(* IEC 61131-3 sources: AXOpen/src/components.festo.drives/ctrl/src/AxoCmmtAs (part 3) *)

                        MC_TorqueControlPositionLimit_PV :=  PositionLimit;
                        MC_TorqueControlVelocity_PV      :=  Velocity;
                        MC_TorqueControlAcceleration_PV  :=  Acceleration;
                        MC_TorqueControlDeceleration_PV  :=  Deceleration;
                        MC_TorqueControlJerk_PV          :=  Jerk;
                        MC_TorqueControlDirection_PV     :=  Direction;
                        MC_TorqueControlTorque_PV        :=  Torque;
                        MC_TorqueControlTorqueRamp_PV    :=  TorqueRamp;
                        State := UINT#120;
                    END_IF;
                END_IF;
                IF State = UINT#120 THEN
                    Busy := TRUE;
                    Active := TRUE;
                    IF MC_TorqueControlPositiveDirectionA AND THIS.ActualPosition >= MC_TorqueControlPositionLimit_PV THEN
                        State := UINT#129;
                        Messenger.Activate(         UINT#1538, eAxoMessageCategory#ProgrammingError);
                        MC_TorqueControlErrorID :=  DINT#1538;
                    ELSIF NOT MC_TorqueControlPositiveDirectionA AND THIS.ActualPosition <= MC_TorqueControlPositionLimit_PV THEN
                        State := UINT#129;
                        Messenger.Activate(         UINT#1539, eAxoMessageCategory#ProgrammingError);
                        MC_TorqueControlErrorID :=  DINT#1539;
                    ELSE
                        State := UINT#121;
                    END_IF;
                END_IF;
                //Writing PNU 12168 Clamping torque
                IF State = UINT#121 THEN
                    Busy := TRUE;
                    Active := TRUE;
                    Parametrization.Inputs.Enable := TRUE;
                    Parametrization.Inputs.ReadWrite   := TRUE;
                    Parametrization.Inputs.ParameterNo := 12168;
                    Parametrization.Inputs.Subindex    := 0;
                    Parametrization.Inputs.AxisNo  := BYTE#1;
                    Parametrization.Inputs.HardwareId  := _AxisReference^.HWIDs.HW_ModuleAccessPoint;
                    Parametrization.Inputs.ValueWriteREAL := TO_REAL(MC_TorqueControlTorque_PV * ScalingConstantRequiredTorque);
                    IF Parametrization.Outputs.Done AND NOT Parametrization.Outputs.Error THEN
                        Parametrization.Inputs.Enable := FALSE;
                        Parametrization.Inputs.ReadWrite   := FALSE;
                        State := UINT#122;
                        RETURN;
                    END_IF;
                    IF Parametrization.Outputs.Error THEN
                        Messenger.Activate(         UINT#1540, eAxoMessageCategory#Error);
                        MC_TorqueControlErrorID :=  DINT#1540;
                        Parametrization.Inputs.Enable := FALSE;
                        Parametrization.Inputs.ReadWrite   := FALSE;
                        State := UINT#129;
                    END_IF;
                END_IF;
                //Writing PNU 11822 Default value torque rise ramp torque
                IF State = UINT#122 THEN
                    Busy := TRUE;
                    Active := TRUE;
                    Parametrization.Inputs.Enable := TRUE;
                    Parametrization.Inputs.ReadWrite   := TRUE;
                    Parametrization.Inputs.ParameterNo := 11822;
                    Parametrization.Inputs.Subindex    := 0;
                    Parametrization.Inputs.AxisNo  := BYTE#1;
                    Parametrization.Inputs.HardwareId  := _AxisReference^.HWIDs.HW_ModuleAccessPoint;
                    Parametrization.Inputs.ValueWriteREAL := TO_REAL(MC_TorqueControlTorqueRamp_PV);
                    IF Parametrization.Outputs.Done AND NOT Parametrization.Outputs.Error THEN
                        Parametrization.Inputs.Enable := FALSE;
                        Parametrization.Inputs.ReadWrite   := FALSE;
                        State := UINT#123;
                        RETURN;
                    END_IF;
                    IF Parametrization.Outputs.Error THEN
                        Messenger.Activate(         UINT#1540, eAxoMessageCategory#Error);
                        MC_TorqueControlErrorID :=  DINT#1540;
                        Parametrization.Inputs.Enable := FALSE;
                        Parametrization.Inputs.ReadWrite   := FALSE;
                        State := UINT#129;
                    END_IF;
                END_IF;
                //Writing PNU 12327 Jerk
                IF State = UINT#123 THEN
                    Busy := TRUE;
                    Active := TRUE;
                    Parametrization.Inputs.Enable := TRUE;
                    Parametrization.Inputs.ReadWrite   := TRUE;
                    Parametrization.Inputs.ParameterNo := 12327;
                    Parametrization.Inputs.Subindex    := 0;
                    Parametrization.Inputs.AxisNo  := BYTE#1;
                    Parametrization.Inputs.HardwareId  := _AxisReference^.HWIDs.HW_ModuleAccessPoint;
                    Parametrization.Inputs.ValueWriteREAL := TO_REAL(MC_TorqueControlJerk_PV  * ScalingConstantRequiredJerk * _AxisReference^.Data.OverrideJerkFactor);
                    IF Parametrization.Outputs.Done AND NOT Parametrization.Outputs.Error THEN
                        Parametrization.Inputs.Enable := FALSE;
                        Parametrization.Inputs.ReadWrite   := FALSE;
                        State := UINT#124;
                        RETURN;
                    END_IF;
                    IF Parametrization.Outputs.Error THEN
                        Messenger.Activate(         UINT#1541, eAxoMessageCategory#Error);
                        MC_TorqueControlErrorID :=  DINT#1541;
                        State := UINT#129;
                    END_IF;
                END_IF;

                // //Writing P1.102223.0.0 – Selection of dynamic torque boost → [0] None
                // // PNU 13073.0 - USINT
                // IF State = UINT#1123 THEN
                //     Busy := TRUE;
                //     Active := TRUE;
                //     Parametrization.Inputs.Enable := TRUE;
                //     Parametrization.Inputs.ReadWrite   := TRUE;
                //     Parametrization.Inputs.ParameterNo := 13073;
                //     Parametrization.Inputs.Subindex    := 0;
                //     Parametrization.Inputs.AxisNo  := BYTE#1;
                //     Parametrization.Inputs.HardwareId  := _AxisReference^.HWIDs.HW_ModuleAccessPoint;
                //     Parametrization.Inputs.ValueWriteLINT := LINT#0;
                //     IF Parametrization.Outputs.Done AND NOT Parametrization.Outputs.Error THEN
                //         Parametrization.Inputs.Enable := FALSE;
                //         Parametrization.Inputs.ReadWrite   := FALSE;
                //         State := UINT#124;
                //         RETURN;
                //     END_IF;
                //     IF Parametrization.Outputs.Error THEN
                //         Messenger.Activate(         UINT#1543, eAxoMessageCategory#Error);
                //         MC_TorqueControlErrorID :=  DINT#1543;
                //         State := UINT#129;
                //     END_IF;
                // END_IF;

                IF State = UINT#124 THEN
                    Busy := TRUE;
                    Active := TRUE;
                    Parametrization.Inputs.Enable := FALSE;
                    Parametrization.Inputs.ReadWrite   := FALSE;
                    IF  NOT Parametrization.Outputs.Done THEN
                        State := UINT#125;
                    END_IF;
                END_IF;
                //Executing movement
                IF State = UINT#125 THEN
                    Busy := TRUE;
                    Active := TRUE;
                    _AxisReference^.Telegram111_Out.POS_STW1.MDI_Activate := TRUE;
                    _AxisReference^.Telegram111_Out.POS_STW1.MDI_MOD := FALSE;
                    _AxisReference^.Telegram111_Out.POS_STW1.SetupMode := FALSE;
                    _AxisReference^.Telegram111_Out.STW2.TravelToFixStop := TRUE;
                    _AxisReference^.Telegram111_Out.STW1.activateTraversing := TRUE;

                    IF _AxisReference^.Telegram111_In.ZSW1.acknowledgeTraversingBlockActivated THEN
                        _AxisReference^.Telegram111_Out.STW1.activateTraversing := FALSE;
                        State := UINT#126;
                    END_IF;
                END_IF;

                IF (State = UINT#126 OR State = UINT#127 OR MC_TorqueControlContinuousUpdate_SV) AND
                    _AxisReference^.Telegram111_In.POS_ZSW2.%X13 THEN
                    InTorque := MC_TorqueControlTorqueWindowTimer.OnDelay(  Parent := THIS,
                                                                            inSignal := ActualTorque >= MC_TorqueControlTorqueWindowMin AND ActualTorque <= MC_TorqueControlTorqueWindowMax,
                                                                            TimeDelay := _AxisReference^.Config.InTorqueWindowTime);
                ELSE
                    MC_TorqueControlTorqueWindowTimer.OnDelay(  Parent := THIS,inSignal := FALSE,TimeDelay := LT#0s);
                    InTorque := FALSE;
                END_IF;

                IF State = UINT#126 THEN
                    IF NOT MC_TorqueControlContinuousUpdate_SV THEN
                        State := UINT#127;
                    END_IF;
                END_IF;
                IF State = UINT#127 THEN
                    MC_TorqueControlCycle := ULINT#0;
                END_IF;
                IF State = UINT#128 THEN
                    CommandAborted := TRUE;
                END_IF;
                IF State = UINT#129 THEN
                    MC_TorqueControlCycle := ULINT#0;
                    Error := TRUE;
                END_IF;

                // ! IT IS NOT STABLE !
                // IF (State=UINT#126 OR State =UINT#127) AND _AxisReference^.Telegram111_In.ZSW1.targetPosReached THEN
                //     Messenger.Activate(         UINT#1542, eAxoMessageCategory#ProgrammingError);
                //     MC_TorqueControlErrorID :=  DINT#1542;
                //     State := UINT#129;
                // END_IF;

                IF State>=UINT#120 AND State<UINT#127 THEN
                    IF MC_TorqueControlContinuousUpdate_SV AND (
                        MC_TorqueControlTorque_PV        <>  Torque OR
                        MC_TorqueControlTorqueRamp_PV    <>  TorqueRamp OR
                        MC_TorqueControlPositionLimit_PV <>  PositionLimit OR
                        MC_TorqueControlVelocity_PV      <>  Velocity OR
                        MC_TorqueControlAcceleration_PV  <>  Acceleration OR
                        MC_TorqueControlDeceleration_PV  <>  Deceleration OR
                        MC_TorqueControlJerk_PV          <>  Jerk OR
                        MC_TorqueControlDirection_PV     <>  Direction ) THEN
                        _AxisReference^.Telegram111_Out.STW1.activateTraversing := FALSE;
                        IF NOT _AxisReference^.Telegram111_In.ZSW1.acknowledgeTraversingBlockActivated THEN
                            State := UINT#120;
                        END_IF;
                    END_IF;
                    IF NOT _AxisReference^.Telegram111_In.ZSW1.operationEnabled THEN
                        State := UINT#128;
                    ELSIF _AxisReference^.Telegram111_In.ZSW1.faultPresent THEN
                        IF MC_TorqueControlErrorID = DINT#0 THEN
                            MC_TorqueControlErrorID := TO_DINT(_AxisReference^.Telegram111_In.Fault_Code);
                        END_IF;
                        State := UINT#129;
                    ELSIF _AxisReference^.Data.Cycle <> MC_TorqueControlCycle THEN
                        _AxisReference^.Data.Cycle := _AxisReference^.Data.Cycle - ULINT#1;
                        State := UINT#128;
                    END_IF;
                END_IF;
                THIS.UpdateOutputs(AxisRef);
            END_IF;

            IF THIS.AxoTorqueControl_Task.DoneReached() THEN
                _AxisReference^.Status.CurrentMotionTaskId := AXOpen.Components.Drives.eAxoMotionTaskId#Axo_Done;
                _AxisReference^.Telegram111_Out.STW1.activateTraversing := FALSE;
                MC_TorqueControlErrorID := DINT#0;
                // MC_TorqueControlCycle := ULINT#0;
                State := UINT#0;
                THIS.UpdateOutputs(AxisRef);
            END_IF;

            IF THIS.AxoTorqueControl_Task.RestoreTriggered() AND State>=UINT#120 AND State<=UINT#129 THEN
                _AxisReference^.Status.CurrentMotionTaskId := AXOpen.Components.Drives.eAxoMotionTaskId#Axo_None;
                _AxisReference^.Telegram111_Out.STW1.activateTraversing := FALSE;
                MC_TorqueControlErrorID := DINT#0;
                MC_TorqueControlCycle := ULINT#0;
                State := UINT#0;
                THIS.UpdateOutputs(AxisRef);
            END_IF;

            ErrorID := MC_TorqueControlErrorID;
            MC_TorqueControlExecute_PV := Execute;
        END_METHOD

        ///<summary>
        /// This method shifts the coordinate system of an axis by manipulating both the set-point position as well as the
        /// actual position of an axis with the same value without any movement caused. (Re-calibration with same following error).
        /// This can be used for instance for a reference situation. This method can also be used during motion without changing
        /// the commanded position, which is now positioned in the shifted coordinate system.
        ///</summary>
        VAR INTERNAL
            MC_SetPositionExecute_PV				: 	BOOL;				//Execute - previous value
            MC_SetPositionErrorID					: 	DINT;
            MC_SetPositionCycle					    : 	ULINT;
            MC_SetPositionActualPosition            : 	LINT;
        END_VAR
        METHOD PUBLIC OVERRIDE MC_SetPosition
            VAR_INPUT
                AxisRef         :   AXOpen.Components.Abstractions.Drives.IAxoAxisReference;
                Execute         :   BOOL;                       //  Start setting position in axis
                Position        :   LREAL;                       //  Position unit [u] (Means ‘Distance’ if ‘Relative’= TRUE)
                Relative        :   BOOL;                       //  ‘Relative’ distance if True, ‘Absolute’ position if False (= Default)
                ExecutionMode   :   AXOpen.Components.Abstractions.Drives.eAxoExecutionMode;          //  Defines the chronological sequence of the method.
            END_VAR
            VAR_OUTPUT
                Done            :   BOOL;                       //  ‘Position’ has new value
                Busy            :   BOOL;                       //  The method is not finished and new output values are to be expected
                Error           :   BOOL;                       //  Signals that an error has occurred within the method
                ErrorID         :   DINT;                       //  Error identification
            END_VAR
            VAR
                _AxisReference :  REF_TO AXOpen.Components.Festo.Drives.AxoCmmtAsAxisReference;
                Dummy : BOOL;
            END_VAR

            _AxisReference ?= AxisRef;

            IF(_AxisReference = NULL) THEN
                Messenger.Activate(     UINT#1550, eAxoMessageCategory#ProgrammingError);
                DriveStatus.Error.Id := UINT#1550;
                RETURN;
            END_IF;

            IF THIS.AxoSetPosition_Task.StartTriggered() THEN
                _AxisReference^.Status.CurrentMotionTaskId := AXOpen.Components.Drives.eAxoMotionTaskId#Axo_SetPosition;
            END_IF;

            IF Execute AND NOT MC_SetPositionExecute_PV AND State = UINT#0 THEN
                _AxisReference^.Data.Cycle := _AxisReference^.Data.Cycle + ULINT#2;
                MC_SetPositionCycle := _AxisReference^.Data.Cycle ;
            END_IF;

            IF Execute THEN
                THIS.UpdateInputs(AxisRef);
                IF State = UINT#0 THEN
                    Busy := TRUE;
                    MC_SetPositionErrorID := DINT#0;
                    _AxisReference^.Telegram111_Out.STW1.StartHoming := FALSE;
                    _AxisReference^.Telegram111_Out.STW1.activateTraversing := FALSE;
                    _AxisReference^.Telegram111_Out.POS_STW1.MDI_MOD := FALSE;
                    _AxisReference^.Telegram111_Out.POS_STW1.PosModulo := FALSE;
                    _AxisReference^.Telegram111_Out.POS_STW1.NegModulo := FALSE;
                    _AxisReference^.Telegram111_Out.POS_STW1.SetupMode := FALSE;
                    _AxisReference^.Telegram111_Out.POS_STW1.MDI_Activate := FALSE;
                    _AxisReference^.Telegram111_Out.POS_STW2.Trackingmode := FALSE;
                    _AxisReference^.Telegram111_Out.POS_STW2.jog_inc := FALSE;
                    _AxisReference^.Telegram111_Out.POS_STW1.travBlockBit0 := FALSE;
                    _AxisReference^.Telegram111_Out.POS_STW1.travBlockBit1 := FALSE;
                    _AxisReference^.Telegram111_Out.POS_STW1.travBlockBit2 := FALSE;
                    _AxisReference^.Telegram111_Out.POS_STW1.travBlockBit3 := FALSE;
                    _AxisReference^.Telegram111_Out.POS_STW1.travBlockBit4 := FALSE;
                    _AxisReference^.Telegram111_Out.POS_STW1.travBlockBit5 := FALSE;
                    _AxisReference^.Telegram111_Out.POS_STW1.travBlockBit6 := FALSE;
                    _AxisReference^.Telegram111_Out.STW2.TravelToFixStop := FALSE;
                    Parametrization.Inputs.Enable := FALSE;
                    State := UINT#130;
                END_IF;
                //Read  PNU 11735 Homing mode
                IF State = UINT#130 THEN
                    Busy := TRUE;
                    Parametrization.Inputs.Enable := TRUE;
                    Parametrization.Inputs.ReadWrite   := FALSE;
                    Parametrization.Inputs.ParameterNo := 11735;//mode
                    Parametrization.Inputs.Subindex    := 0;
                    Parametrization.Inputs.AxisNo  := BYTE#1;
                    Parametrization.Inputs.HardwareId  := _AxisReference^.HWIDs.HW_ModuleAccessPoint;
                    IF Parametrization.Outputs.Done AND NOT Parametrization.Outputs.Error THEN
                        PNU_11735 := Parametrization.Outputs.ValueReadLINT;
                        State := UINT#131;
                    END_IF;
                    IF Parametrization.Outputs.Error THEN
                        Messenger.Activate(         UINT#1551, eAxoMessageCategory#Error);
                        MC_SetPositionErrorID :=    DINT#1551;
                        State := UINT#159;
                    END_IF;
                END_IF;
                IF State = UINT#131 THEN
                    Busy := TRUE;
                    Parametrization.Inputs.Enable := FALSE;
                    IF  NOT Parametrization.Outputs.Done THEN
                        State := UINT#132;
                    END_IF;
                END_IF;
                //Write  PNU 12681 deactivate save zero offset
                IF State = UINT#132 THEN
                    Busy := TRUE;
                    Parametrization.Inputs.Enable := TRUE;
                    Parametrization.Inputs.ReadWrite   := TRUE;
                    Parametrization.Inputs.ParameterNo := 12681;//deactivate save zero offset
                    Parametrization.Inputs.Subindex    := 0;
                    Parametrization.Inputs.AxisNo  := BYTE#1;
                    Parametrization.Inputs.HardwareId  := _AxisReference^.HWIDs.HW_ModuleAccessPoint;
                    Parametrization.Inputs.ValueWriteBOOL := FALSE;
                    IF Parametrization.Outputs.Done AND NOT Parametrization.Outputs.Error THEN
                        State := UINT#133;
                    END_IF;
                    IF Parametrization.Outputs.Error THEN
                        Messenger.Activate(         UINT#1552, eAxoMessageCategory#Error);
                        MC_SetPositionErrorID :=    DINT#1552;
                        State := UINT#159;
                    END_IF;
                END_IF;
                IF State = UINT#133 THEN
                    Busy := TRUE;
                    Parametrization.Inputs.Enable := FALSE;
                    IF  NOT Parametrization.Outputs.Done THEN
                        State := UINT#134;
                    END_IF;
                END_IF;
                //Read PNU 11203 Move to axis zero after homming
                IF State = UINT#134 THEN
                    Busy := TRUE;
                    Parametrization.Inputs.Enable := TRUE;
                    Parametrization.Inputs.ReadWrite   := FALSE;
                    Parametrization.Inputs.ParameterNo := 11203;//Move to axis zero after homming
                    Parametrization.Inputs.Subindex    := 0;
                    Parametrization.Inputs.AxisNo  := BYTE#1;
                    Parametrization.Inputs.HardwareId  := _AxisReference^.HWIDs.HW_ModuleAccessPoint;
                    IF Parametrization.Outputs.Done AND NOT Parametrization.Outputs.Error THEN
                        PNU_11203 := Parametrization.Outputs.ValueReadBool;
                        State := UINT#135;
                    END_IF;
                    IF Parametrization.Outputs.Error THEN
                        Messenger.Activate(         UINT#1553, eAxoMessageCategory#Error);
                        MC_SetPositionErrorID :=    DINT#1553;
                        State := UINT#159;
                    END_IF;
                END_IF;
                IF State = UINT#135 THEN
                    Busy := TRUE;
                    Parametrization.Inputs.Enable := FALSE;
                    IF  NOT Parametrization.Outputs.Done THEN
                        State := UINT#136;
                    END_IF;
                END_IF;
                //Read PNU 11734 Axis zero point offset
                IF State = UINT#136 THEN
                    Busy := TRUE;
                    Parametrization.Inputs.Enable := TRUE;
                    Parametrization.Inputs.ReadWrite   := FALSE;
                    Parametrization.Inputs.ParameterNo := 11734;//Move to axis zero after homming
                    Parametrization.Inputs.Subindex    := 0;
                    Parametrization.Inputs.AxisNo  := BYTE#1;
                    Parametrization.Inputs.HardwareId  := _AxisReference^.HWIDs.HW_ModuleAccessPoint;
                    IF Parametrization.Outputs.Done AND NOT Parametrization.Outputs.Error THEN
                        PNU_11734 := Parametrization.Outputs.ValueReadLINT;
                        State := UINT#137;
                    END_IF;
                    IF Parametrization.Outputs.Error THEN
                        Messenger.Activate(         UINT#1554, eAxoMessageCategory#Error);
                        MC_SetPositionErrorID :=    DINT#1554;
                        State := UINT#159;
                    END_IF;
                END_IF;
                IF State = UINT#137 THEN
                    Busy := TRUE;
                    Parametrization.Inputs.Enable := FALSE;
                    IF  NOT Parametrization.Outputs.Done THEN
                        State := UINT#138;
                    END_IF;
                END_IF;
                //Write PNU 11203 deactivate Move to axis zero after homming
                IF State = UINT#138 THEN
                    Busy := TRUE;
                    Parametrization.Inputs.Enable := TRUE;
                    Parametrization.Inputs.ReadWrite   := TRUE;
                    Parametrization.Inputs.ParameterNo := 11203;//Move to axis zero after homming
                    Parametrization.Inputs.Subindex    := 0;
                    Parametrization.Inputs.AxisNo  := BYTE#1;
                    Parametrization.Inputs.HardwareId  := _AxisReference^.HWIDs.HW_ModuleAccessPoint;
                    Parametrization.Inputs.ValueWriteBOOL := FALSE;
                    IF Parametrization.Outputs.Done AND NOT Parametrization.Outputs.Error THEN
                        State := UINT#139;
                    END_IF;
                    IF Parametrization.Outputs.Error THEN
                        Messenger.Activate(         UINT#1555, eAxoMessageCategory#Error);
                        MC_SetPositionErrorID :=    DINT#1555;
                        State := UINT#159;
                    END_IF;
                END_IF;
                IF State = UINT#139 THEN
                    Busy := TRUE;
                    Parametrization.Inputs.Enable := FALSE;
                    MC_SetPositionActualPosition :=  TO_LINT(ActualPosition * -10000000000.0);
                    IF  NOT Parametrization.Outputs.Done THEN
                        State := UINT#140;
                    END_IF;
                END_IF;
                //Write PNU 11734 Axis zero point offset
                IF State = UINT#140 THEN
                    Busy := TRUE;
                    Parametrization.Inputs.Enable := TRUE;
                    Parametrization.Inputs.ReadWrite   := TRUE;
                    Parametrization.Inputs.ParameterNo := 11734;//Move to axis zero after homming
                    Parametrization.Inputs.Subindex    := 0;
                    Parametrization.Inputs.AxisNo  := BYTE#1;
                    Parametrization.Inputs.HardwareId  := _AxisReference^.HWIDs.HW_ModuleAccessPoint;
                    IF Relative THEN
                        Parametrization.Inputs.ValueWriteLINT := MC_SetPositionActualPosition + TO_LINT(Position * -10000000.0);
                    ELSE
                        Parametrization.Inputs.ValueWriteLINT := TO_LINT(Position * -10000000.0);
                    END_IF;
                    IF Parametrization.Outputs.Done AND NOT Parametrization.Outputs.Error THEN
                        State := UINT#141;
                    END_IF;
                    IF Parametrization.Outputs.Error THEN
                        Messenger.Activate(         UINT#1556, eAxoMessageCategory#Error);
                        MC_SetPositionErrorID :=    DINT#1556;
                        State := UINT#159;
                    END_IF;
                END_IF;
                IF State = UINT#141 THEN
                    Busy := TRUE;
                    Parametrization.Inputs.Enable := FALSE;
                    IF  NOT Parametrization.Outputs.Done THEN
                        State := UINT#142;
                    END_IF;
                END_IF;
                //Write  PNU 11735 Homing mode
                IF State = UINT#142 THEN
                    Busy := TRUE;
                    Parametrization.Inputs.Enable := TRUE;
                    Parametrization.Inputs.ReadWrite   := TRUE;
                    Parametrization.Inputs.ParameterNo := 11735;//mode
                    Parametrization.Inputs.Subindex    := 0;
                    Parametrization.Inputs.AxisNo  := BYTE#1;
                    Parametrization.Inputs.HardwareId  := _AxisReference^.HWIDs.HW_ModuleAccessPoint;
                    Parametrization.Inputs.ValueWriteLINT := TO_LINT(37);
                    IF Parametrization.Outputs.Done AND NOT Parametrization.Outputs.Error THEN
                        State := UINT#143;
                    END_IF;
                    IF Parametrization.Outputs.Error THEN
                        Messenger.Activate(         UINT#1557, eAxoMessageCategory#Error);
                        MC_SetPositionErrorID :=    DINT#1557;
                        State := UINT#159;
                    END_IF;
                END_IF;
                IF State = UINT#143 THEN
                    Busy := TRUE;
                    Parametrization.Inputs.Enable := FALSE;
                    IF  NOT Parametrization.Outputs.Done THEN
                        State := UINT#144;
                    END_IF;
                END_IF;
                //Homing started
                IF State = UINT#144 THEN
                    Busy := TRUE;
                    _AxisReference^.Telegram111_Out.STW1.StartHoming := TRUE;
                    IF  NOT _AxisReference^.Telegram111_In.ZSW1.targetPosReached AND NOT _AxisReference^.Telegram111_In.ZSW1.homePosSet THEN
                        State := UINT#145;
                    END_IF;
                END_IF;
                IF State = UINT#145 THEN
                    Busy := TRUE;
                    IF _AxisReference^.Telegram111_In.ZSW1.targetPosReached AND _AxisReference^.Telegram111_In.ZSW1.homePosSet THEN
                        _AxisReference^.Telegram111_Out.STW1.StartHoming := FALSE;
                        State := UINT#146;
                    END_IF;
                END_IF;
                //Write PNU 11203 Move to axis zero after homming
                IF State = UINT#146 THEN
                    Busy := TRUE;
                    Parametrization.Inputs.Enable := TRUE;
                    Parametrization.Inputs.ReadWrite   := TRUE;
                    Parametrization.Inputs.ParameterNo := 11203;//Move to axis zero after homming
                    Parametrization.Inputs.Subindex    := 0;
                    Parametrization.Inputs.AxisNo  := BYTE#1;
                    Parametrization.Inputs.HardwareId  := _AxisReference^.HWIDs.HW_ModuleAccessPoint;
                    Parametrization.Inputs.ValueWriteBool := PNU_11203;
                    IF Parametrization.Outputs.Done AND NOT Parametrization.Outputs.Error THEN
                        State := UINT#147;
                    END_IF;
                    IF Parametrization.Outputs.Error THEN
                        Messenger.Activate(         UINT#1558, eAxoMessageCategory#Error);
                        MC_SetPositionErrorID :=    DINT#1558;
                        State := UINT#159;
                    END_IF;
                END_IF;
                IF State = UINT#147 THEN
                    Busy := TRUE;
                    Parametrization.Inputs.Enable := FALSE;
                    IF  NOT Parametrization.Outputs.Done THEN
                        State := UINT#148;
                    END_IF;
                END_IF;
                //Write PNU 11734 Axis zero point offset
                IF State = UINT#148 THEN
                    Busy := TRUE;
                    Parametrization.Inputs.Enable := TRUE;
                    Parametrization.Inputs.ReadWrite   := TRUE;
                    Parametrization.Inputs.ParameterNo := 11734;//Move to axis zero after homming
                    Parametrization.Inputs.Subindex    := 0;
                    Parametrization.Inputs.AxisNo  := BYTE#1;
                    Parametrization.Inputs.HardwareId  := _AxisReference^.HWIDs.HW_ModuleAccessPoint;
                    Parametrization.Inputs.ValueWriteLINT := PNU_11734;
                    IF Parametrization.Outputs.Done AND NOT Parametrization.Outputs.Error THEN
                         State := UINT#149;
                    END_IF;
                    IF Parametrization.Outputs.Error THEN
                        Messenger.Activate(         UINT#1559, eAxoMessageCategory#Error);
                        MC_SetPositionErrorID :=    DINT#1559;
                        State := UINT#159;
                    END_IF;
                END_IF;
                IF State = UINT#149 THEN
                    Busy := TRUE;
                    Parametrization.Inputs.Enable := FALSE;
                    IF  NOT Parametrization.Outputs.Done THEN
                        State := UINT#150;
                    END_IF;
                END_IF;
                //Write PNU 11735 homming mode
                IF State = UINT#150 THEN
                    Parametrization.Inputs.Enable := TRUE;
                    Parametrization.Inputs.ReadWrite   := TRUE;
                    Parametrization.Inputs.ParameterNo := 11735;
                    Parametrization.Inputs.Subindex    := 0;
                    Parametrization.Inputs.AxisNo  := BYTE#1;
                    Parametrization.Inputs.HardwareId  := _AxisReference^.HWIDs.HW_ModuleAccessPoint;
                    Parametrization.Inputs.ValueWriteLINT := PNU_11735;
                    IF Parametrization.Outputs.Done AND NOT Parametrization.Outputs.Error THEN
                        State := UINT#151;
                    END_IF;
                    IF Parametrization.Outputs.Error THEN
                        Messenger.Activate(         UINT#1560, eAxoMessageCategory#Error);
                        MC_SetPositionErrorID :=    DINT#1560;
                        State := UINT#159;
                   END_IF;
                END_IF;
                IF State = UINT#151 THEN
                    Busy := TRUE;
                    Parametrization.Inputs.Enable := FALSE;
                    IF  NOT Parametrization.Outputs.Done THEN
                        State := UINT#152;
                    END_IF;
                END_IF;
                IF State = UINT#152 THEN
                    Busy := TRUE;
                    IF TRUE THEN
                        State := UINT#153;
                    END_IF;
                END_IF;
                IF State = UINT#153 THEN
                    Busy := TRUE;
                    IF TRUE THEN
                        State := UINT#154;
                    END_IF;
                END_IF;
                IF State = UINT#154 THEN
                    Busy := TRUE;
                    IF TRUE THEN
                        State := UINT#155;
                    END_IF;
                END_IF;
                IF State = UINT#155 THEN
                    Busy := TRUE;
                    IF TRUE THEN
                        State := UINT#156;
                    END_IF;
                END_IF;
                IF State = UINT#156 THEN
                    Busy := TRUE;
                    IF TRUE THEN
                        State := UINT#157;
                    END_IF;
                END_IF;
                IF State = UINT#157 THEN
                    _AxisReference^.Telegram111_Out.STW1.StartHoming := FALSE;
                    Done := TRUE;
                    MC_SetPositionCycle := ULINT#0;
                END_IF;
                IF State = UINT#158 THEN
                    _AxisReference^.Telegram111_Out.STW1.StartHoming := FALSE;
                END_IF;
                IF State = UINT#159 THEN
                    _AxisReference^.Telegram111_Out.STW1.StartHoming := FALSE;
                    MC_SetPositionCycle := ULINT#0;
                    Error := TRUE;
                END_IF;

                IF State>=UINT#130 AND State<UINT#157 THEN
                    IF NOT _AxisReference^.Telegram111_In.ZSW1.operationEnabled THEN
                        State := UINT#158;
                    ELSIF _AxisReference^.Telegram111_In.ZSW1.faultPresent THEN
                        IF MC_SetPositionErrorID = DINT#0 THEN
                            MC_SetPositionErrorID := TO_DINT(_AxisReference^.Telegram111_In.Fault_Code);
                        END_IF;
                        State := UINT#159;
                    ELSIF _AxisReference^.Data.Cycle <> MC_SetPositionCycle THEN
                        _AxisReference^.Data.Cycle := _AxisReference^.Data.Cycle - ULINT#1;
                        State := UINT#158;
                    END_IF;
                END_IF;
            END_IF;

            IF THIS.AxoSetPosition_Task.DoneReached() THEN
                _AxisReference^.Status.CurrentMotionTaskId := AXOpen.Components.Drives.eAxoMotionTaskId#Axo_Done;
                MC_SetPositionErrorID := DINT#0;
                // MC_SetPositionCycle := ULINT#0;
                Parametrization.Inputs.Enable := FALSE;
                Parametrization.Inputs.ReadWrite   := FALSE;
                State := UINT#0;
                THIS.UpdateOutputs(AxisRef);
            END_IF;
            IF THIS.AxoSetPosition_Task.RestoreTriggered() AND State>=UINT#130 AND State<=UINT#159 THEN
                _AxisReference^.Status.CurrentMotionTaskId := AXOpen.Components.Drives.eAxoMotionTaskId#Axo_None;
                MC_SetPositionErrorID := DINT#0;
                MC_SetPositionCycle := ULINT#0;
                Parametrization.Inputs.Enable := FALSE;
                Parametrization.Inputs.ReadWrite   := FALSE;
                State := UINT#0;
                THIS.UpdateOutputs(AxisRef);
            END_IF;

            ErrorID := MC_SetPositionErrorID;
            MC_SetPositionExecute_PV := Execute;
        END_METHOD

        ///<summary>
        /// This method sets the values of override for the whole axis, and all functions that are working on that axis. The override
        /// parameters contribute as a factor to the calculation of the commanded velocity, acceleration and jerk of the motion.
        ///<summary>
        METHOD PUBLIC OVERRIDE MC_SetOverride
            VAR_INPUT
                AxisRef         :   AXOpen.Components.Abstractions.Drives.IAxoAxisReference;
                Enable          :   BOOL;                       //  If SET, it writes the value of the override factor continuously. If RESET it should keep the last value.
                VelocityFactor  :   LREAL;                      //  New override factor for the velocity
                AccelerationFactor:   LREAL;                    //  New override factor for the acceleration/deceleration
                JerkFactor      :   LREAL;                      //  New override factor for the jer
            END_VAR
            VAR_OUTPUT
                Enabled         :   BOOL;                       //  Signals that the override factor(s) is (are) set successfully
                Busy            :   BOOL;                       //  The method is not finished and new output values are to be expected
                Error           :   BOOL;                       //  Signals that an error has occurred within the method
                ErrorID         :   DINT;                       //  Error identification
            END_VAR
            VAR
                _AxisReference :  REF_TO AXOpen.Components.Festo.Drives.AxoCmmtAsAxisReference;
                Dummy : BOOL;
            END_VAR

            _AxisReference ?= AxisRef;

            IF(_AxisReference = NULL) THEN
                Messenger.Activate(     UINT#1570, eAxoMessageCategory#ProgrammingError);
                DriveStatus.Error.Id := UINT#1570;
                RETURN;
            END_IF;

            Messenger.ActivateOnCondition(ULINT#1571, Enable AND  (VelocityFactor <= 0.0 OR  VelocityFactor >= 2.0), eAxoMessageCategory#ProgrammingError);
            Messenger.ActivateOnCondition(ULINT#1572, Enable AND  (AccelerationFactor <= 0.0 OR  AccelerationFactor > 1.0), eAxoMessageCategory#ProgrammingError);
            Messenger.ActivateOnCondition(ULINT#1573, Enable AND  (JerkFactor <= 0.0 OR JerkFactor > 1.0), eAxoMessageCategory#ProgrammingError);

            IF Enable THEN
                Busy := TRUE;
                IF VelocityFactor <= 0.0 OR  VelocityFactor >= 2.0 OR AccelerationFactor <= 0.0 OR  AccelerationFactor > 1.0 OR JerkFactor <= 0.0 OR  JerkFactor > 1.0 THEN
                    Error := TRUE;
                ELSE
                    _AxisReference^.Data.OverrideVelocityFactor := VelocityFactor;
                    _AxisReference^.Data.OverrideAccelerationFactor := AccelerationFactor;
                    _AxisReference^.Data.OverrideJerkFactor := JerkFactor;
                    _AxisReference^.Telegram111_Out.Override_ := TO_WORD(TO_INT(16384.0/VelocityFactor));
                    THIS.UpdateOutputs(AxisRef);
                    Enabled	:= TRUE;
                END_IF;
            END_IF;
        END_METHOD

        ///<summary>
        /// This method returns the value of a vendor specific parameter. The returned Value has to be converted to Real
        /// if necessary. If not possible, the vendor has to supply a vendor specific method to read the parameter.
        ///</summary>
        VAR INTERNAL
            MC_ReadParameterEnable_PV       : 	BOOL := FALSE;		//Enable - previous value
            MC_ReadParameterErrorID         : 	DINT;
            MC_ReadParameterCycle			: 	ULINT;
            MC_ReadParameterValue			: 	LINT;
            MC_ReadParameterValid			: 	BOOL;
        END_VAR
        METHOD PUBLIC OVERRIDE MC_ReadParameter
            VAR_INPUT
                AxisRef         :   AXOpen.Components.Abstractions.Drives.IAxoAxisReference;
                Enable          :   BOOL;                       //  Get the value of the parameter continuously while enabled
                ParameterNumber :   DINT;                       //  Number of the parameter. One can also use symbolic parameter names which are declared as VAR CONST.
            END_VAR
            VAR_OUTPUT
                Valid           :   BOOL;                       //  A valid output is available at the method
                Busy            :   BOOL;                       //  The method is not finished and new output values are to be expected
                Error           :   BOOL;                       //  Signals that an error has occurred within the method
                ErrorID         :   DINT;                       //  Error identification
                Value           :   LINT;                       //  Value of the specified parameter in the datatype, as specified by the vendor
            END_VAR
            VAR
                _AxisReference :  REF_TO AXOpen.Components.Festo.Drives.AxoCmmtAsAxisReference;
                Dummy : BOOL;
            END_VAR

            _AxisReference ?= AxisRef;

            IF(_AxisReference = NULL) THEN
                Messenger.Activate(     UINT#1580, eAxoMessageCategory#ProgrammingError);
                DriveStatus.Error.Id := UINT#1580;
                RETURN;
            END_IF;

            IF Enable AND NOT MC_ReadParameterEnable_PV AND State = UINT#0 THEN
                _AxisReference^.Status.CurrentMotionTaskId := AXOpen.Components.Drives.eAxoMotionTaskId#Axo_ReadParameter;
                _AxisReference^.Data.Cycle := _AxisReference^.Data.Cycle + ULINT#2;
                MC_ReadParameterCycle := _AxisReference^.Data.Cycle ;
            END_IF;

            IF Enable THEN
                IF State = UINT#0 THEN
                    Busy := TRUE;
                    MC_ReadParameterErrorID := DINT#0;
                    Parametrization.Inputs.Enable := FALSE;
                    State := UINT#160;
                END_IF;
                IF State = UINT#160 THEN
                    Busy := TRUE;
                    Parametrization.Inputs.Enable := TRUE;
                    Parametrization.Inputs.ReadWrite   := FALSE;
                    Parametrization.Inputs.ParameterNo := TO_INT(ParameterNumber);
                    Parametrization.Inputs.Subindex    := 0;
                    Parametrization.Inputs.AxisNo  := BYTE#1;
                    Parametrization.Inputs.HardwareId  := _AxisReference^.HWIDs.HW_ModuleAccessPoint;
                    IF Parametrization.Outputs.Done AND NOT Parametrization.Outputs.Error THEN
                        MC_ReadParameterValid := TRUE;
                        MC_ReadParameterValue := Parametrization.Outputs.ValueReadLINT;
                        State := UINT#161;
                    END_IF;
                    IF Parametrization.Outputs.Error THEN
                        Messenger.Activate(         UINT#1581, eAxoMessageCategory#Error);
                        MC_ReadParameterErrorID :=  DINT#1581;
                        State := UINT#169;
                    END_IF;
                END_IF;
                IF State = UINT#161 THEN
                    Busy := TRUE;
                    Parametrization.Inputs.Enable := FALSE;
                    Parametrization.Inputs.ReadWrite   := FALSE;
                    IF  NOT Parametrization.Outputs.Done THEN
                        State := UINT#160;
                    END_IF;
                END_IF;
                IF State = UINT#169 THEN
                    Error := TRUE;
                END_IF;

                IF State>=UINT#160 AND State<UINT#167 THEN
                    IF _AxisReference^.Data.Cycle <> MC_ReadParameterCycle THEN
                        _AxisReference^.Data.Cycle := _AxisReference^.Data.Cycle - ULINT#1;
                        State := UINT#169;
                    END_IF;
                END_IF;
            END_IF;

            IF NOT Enable AND MC_ReadParameterEnable_PV  THEN
                _AxisReference^.Status.CurrentMotionTaskId := AXOpen.Components.Drives.eAxoMotionTaskId#Axo_None;
                MC_ReadParameterErrorID := DINT#0;
                MC_ReadParameterCycle := ULINT#0;
                MC_ReadParameterValid := FALSE;
                MC_ReadParameterValue := LINT#0;
                State := UINT#0;
            END_IF;

            ErrorID := MC_ReadParameterErrorID;
            Valid := MC_ReadParameterValid;
            Value := MC_ReadParameterValue;
            MC_ReadParameterEnable_PV := Enable;
        END_METHOD

        ///<summary>
        /// This method returns the value of a vendor specific parameter with datatype REAL.
        ///</summary>
        VAR INTERNAL
            MC_ReadRealParameterEnable_PV       : 	BOOL := FALSE;		//Enable - previous value
            MC_ReadRealParameterErrorID         : 	DINT;
            MC_ReadRealParameterCycle			: 	ULINT;
            MC_ReadRealParameterValue			: 	REAL;
            MC_ReadRealParameterValid			: 	BOOL;
        END_VAR
        METHOD PUBLIC OVERRIDE MC_ReadRealParameter
            VAR_INPUT
                AxisRef         :   AXOpen.Components.Abstractions.Drives.IAxoAxisReference;
                Enable          :   BOOL;                       //  Get the value of the parameter continuously while enabled
                ParameterNumber :   DINT;                       //  Number of the parameter. One can also use symbolic parameter names which are declared as VAR CONST.
            END_VAR
            VAR_OUTPUT
                Valid           :   BOOL;                       //  A valid output is available at the method
                Busy            :   BOOL;                       //  The method is not finished and new output values are to be expected
                Error           :   BOOL;                       //  Signals that an error has occurred within the method
                ErrorID         :   DINT;                       //  Error identification
                Value           :   REAL;                       //  Value of the specified parameter in the datatype, as specified by the vendor
            END_VAR
            VAR
                _AxisReference :  REF_TO AXOpen.Components.Festo.Drives.AxoCmmtAsAxisReference;
                Dummy : BOOL;
            END_VAR

            _AxisReference ?= AxisRef;

            IF(_AxisReference = NULL) THEN
                Messenger.Activate(     UINT#1590, eAxoMessageCategory#ProgrammingError);
                DriveStatus.Error.Id := UINT#1590;
                RETURN;
            END_IF;

            IF Enable AND NOT MC_ReadRealParameterEnable_PV AND State = UINT#0 THEN
                _AxisReference^.Status.CurrentMotionTaskId := AXOpen.Components.Drives.eAxoMotionTaskId#Axo_ReadRealParameter;
                _AxisReference^.Data.Cycle := _AxisReference^.Data.Cycle + ULINT#2;
                MC_ReadRealParameterCycle := _AxisReference^.Data.Cycle ;
            END_IF;

            IF Enable THEN
                IF State = UINT#0 THEN
                    Busy := TRUE;
                    MC_ReadRealParameterErrorID := DINT#0;
                    Parametrization.Inputs.Enable := FALSE;
                    State := UINT#170;
                END_IF;
                IF State = UINT#170 THEN
                    Busy := TRUE;
                    Parametrization.Inputs.Enable := TRUE;
                    Parametrization.Inputs.ReadWrite   := FALSE;
                    Parametrization.Inputs.ParameterNo := TO_INT(ParameterNumber);
                    Parametrization.Inputs.Subindex    := 0;
                    Parametrization.Inputs.AxisNo  := BYTE#1;
                    Parametrization.Inputs.HardwareId  := _AxisReference^.HWIDs.HW_ModuleAccessPoint;
                    IF Parametrization.Outputs.Done AND NOT Parametrization.Outputs.Error THEN
                        MC_ReadRealParameterValid := TRUE;
                        MC_ReadRealParameterValue := Parametrization.Outputs.ValueReadREAL;
                        State := UINT#171;
                    END_IF;
                    IF Parametrization.Outputs.Error THEN
                        Messenger.Activate(             UINT#1591, eAxoMessageCategory#Error);
                        MC_ReadRealParameterErrorID :=  DINT#1591;
                        State := UINT#179;
                    END_IF;
                END_IF;
                IF State = UINT#171 THEN
                    Busy := TRUE;
                    Parametrization.Inputs.Enable := FALSE;
                    Parametrization.Inputs.ReadWrite   := FALSE;
                    IF  NOT Parametrization.Outputs.Done THEN
                        State := UINT#170;
                    END_IF;
                END_IF;
                IF State = UINT#179 THEN
                    Error := TRUE;
                END_IF;

                IF State>=UINT#170 AND State<UINT#177 THEN
                    IF _AxisReference^.Data.Cycle <> MC_ReadRealParameterCycle THEN
                        _AxisReference^.Data.Cycle := _AxisReference^.Data.Cycle - ULINT#1;
                        State := UINT#179;
                    END_IF;
                END_IF;
            END_IF;

            IF NOT Enable AND MC_ReadRealParameterEnable_PV  THEN
                _AxisReference^.Status.CurrentMotionTaskId := AXOpen.Components.Drives.eAxoMotionTaskId#Axo_None;
                MC_ReadRealParameterErrorID := DINT#0;
                MC_ReadRealParameterCycle := ULINT#0;
                MC_ReadRealParameterValid := FALSE;
                MC_ReadRealParameterValue := REAL#0.0;
                State := UINT#0;
            END_IF;

            ErrorID := MC_ReadRealParameterErrorID;
            Valid := MC_ReadRealParameterValid;
            Value := MC_ReadRealParameterValue;
            MC_ReadRealParameterEnable_PV := Enable;
        END_METHOD

        ///<summary>
        /// This method returns the value of a vendor specific parameter with datatype BOOL.
        ///</summary>
        VAR INTERNAL
            MC_ReadBoolParameterEnable_PV       : 	BOOL := FALSE;		//Enable - previous value
            MC_ReadBoolParameterErrorID         : 	DINT;
            MC_ReadBoolParameterCycle			: 	ULINT;
            MC_ReadBoolParameterValue			: 	BOOL;
            MC_ReadBoolParameterValid			: 	BOOL;
        END_VAR
        METHOD PUBLIC OVERRIDE MC_ReadBoolParameter
            VAR_INPUT
                AxisRef         :   AXOpen.Components.Abstractions.Drives.IAxoAxisReference;
                Enable          :   BOOL;                       //  Get the value of the parameter continuously while enabled
                ParameterNumber :   DINT;                       //  Number of the parameter. One can also use symbolic parameter names which are declared as VAR CONST.
            END_VAR
            VAR_OUTPUT
                Valid           :   BOOL;                       //  A valid output is available at the method
                Busy            :   BOOL;                       //  The method is not finished and new output values are to be expected
                Error           :   BOOL;                       //  Signals that an error has occurred within the method
                ErrorID         :   DINT;                       //  Error identification
                Value           :   BOOL;                       //  Value of the specified parameter in the datatype, as specified by the vendor
            END_VAR
            VAR
                _AxisReference :  REF_TO AXOpen.Components.Festo.Drives.AxoCmmtAsAxisReference;
                Dummy : BOOL;
            END_VAR
            RETURN;

            _AxisReference ?= AxisRef;

            IF(_AxisReference = NULL) THEN
                Messenger.Activate(     UINT#1600, eAxoMessageCategory#ProgrammingError);
                DriveStatus.Error.Id := UINT#1600;
                RETURN;
            END_IF;

            IF Enable AND NOT MC_ReadBoolParameterEnable_PV AND State = UINT#0 THEN
                _AxisReference^.Status.CurrentMotionTaskId := AXOpen.Components.Drives.eAxoMotionTaskId#Axo_ReadBoolParameter;
                _AxisReference^.Data.Cycle := _AxisReference^.Data.Cycle + ULINT#2;
                MC_ReadBoolParameterCycle := _AxisReference^.Data.Cycle ;
            END_IF;

            IF Enable THEN
                IF State = UINT#0 THEN
                    Busy := TRUE;
                    MC_ReadBoolParameterErrorID := DINT#0;
                    Parametrization.Inputs.Enable := FALSE;
                    State := UINT#180;
                END_IF;
                IF State = UINT#180 THEN
                    Busy := TRUE;
                    Parametrization.Inputs.Enable := TRUE;
                    Parametrization.Inputs.ReadWrite   := FALSE;
                    Parametrization.Inputs.ParameterNo := TO_INT(ParameterNumber);
                    Parametrization.Inputs.Subindex    := 0;
                    Parametrization.Inputs.AxisNo  := BYTE#1;
                    Parametrization.Inputs.HardwareId  := _AxisReference^.HWIDs.HW_ModuleAccessPoint;
                    IF Parametrization.Outputs.Done AND NOT Parametrization.Outputs.Error THEN
                        MC_ReadBoolParameterValid := TRUE;
                        MC_ReadBoolParameterValue := Parametrization.Outputs.ValueReadBOOL;
                        State := UINT#181;
                    END_IF;
                    IF Parametrization.Outputs.Error THEN
                        Messenger.Activate(             UINT#1601, eAxoMessageCategory#Error);
                        MC_ReadBoolParameterErrorID :=  DINT#1601;
                        State := UINT#189;
                    END_IF;
                END_IF;
                IF State = UINT#181 THEN
                    Busy := TRUE;
                    Parametrization.Inputs.Enable := FALSE;
                    Parametrization.Inputs.ReadWrite   := FALSE;
                    IF  NOT Parametrization.Outputs.Done THEN
                        State := UINT#180;
                    END_IF;
                END_IF;
                IF State = UINT#189 THEN
                    Error := TRUE;
                END_IF;

                IF State>=UINT#180 AND State<UINT#187 THEN
                    IF _AxisReference^.Data.Cycle <> MC_ReadBoolParameterCycle THEN
                        _AxisReference^.Data.Cycle := _AxisReference^.Data.Cycle - ULINT#1;
                        State := UINT#189;
                    END_IF;
                END_IF;
            END_IF;

            IF NOT Enable AND MC_ReadBoolParameterEnable_PV  THEN
                _AxisReference^.Status.CurrentMotionTaskId := AXOpen.Components.Drives.eAxoMotionTaskId#Axo_None;
                MC_ReadBoolParameterErrorID := DINT#0;
                MC_ReadBoolParameterCycle := ULINT#0;
                MC_ReadBoolParameterValid := FALSE;
                MC_ReadBoolParameterValue := FALSE;
                State := UINT#0;
            END_IF;

            ErrorID := MC_ReadBoolParameterErrorID;
            Valid := MC_ReadBoolParameterValid;
            Value := MC_ReadBoolParameterValue;
            MC_ReadBoolParameterEnable_PV := Enable;

        END_METHOD

        ///<summary>
        /// This method modifies the value of a vendor specific parameter.
        ///</summary>
        VAR INTERNAL
            MC_WriteParameterExecute_PV     : 	BOOL := FALSE;		//Enable - previous value
            MC_WriteParameterErrorID        : 	DINT;
            MC_WriteParameterCycle			: 	ULINT;
        END_VAR
        METHOD PUBLIC OVERRIDE MC_WriteParameter
            VAR_INPUT
                AxisRef         :   AXOpen.Components.Abstractions.Drives.IAxoAxisReference;
                Execute         :   BOOL;                       //  Write the value of the parameter at rising edge
                ParameterNumber :   DINT;                       //  Number of the parameter (correspondence between number andparameter is specified in the table above)
                Value           :   LINT;                       //  New value of the specified parameter
                ExecutionMode   :   AXOpen.Components.Abstractions.Drives.eAxoExecutionMode;          //  Defines the chronological sequence of the method.
            END_VAR
            VAR_OUTPUT
                Done            :   BOOL;                       //  Parameter successfully written
                Busy            :   BOOL;                       //  The method is not finished and new output values are to be expected.
                Error           :   BOOL;                       //  Signals that an error has occurred within the method
                ErrorID         :   DINT;                       //  Error identification
            END_VAR
            VAR
                _AxisReference :  REF_TO AXOpen.Components.Festo.Drives.AxoCmmtAsAxisReference;
                Dummy : BOOL;
            END_VAR

            _AxisReference ?= AxisRef;

            IF(_AxisReference = NULL) THEN
                Messenger.Activate(     UINT#1610, eAxoMessageCategory#ProgrammingError);
                DriveStatus.Error.Id := UINT#1610;
                RETURN;
            END_IF;

            IF THIS.AxoWriteParameter_Task.StartTriggered()  THEN
                _AxisReference^.Status.CurrentMotionTaskId := AXOpen.Components.Drives.eAxoMotionTaskId#Axo_WriteParameter;
            END_IF;

            IF Execute AND NOT MC_WriteParameterExecute_PV AND State = UINT#0 THEN
                _AxisReference^.Data.Cycle := _AxisReference^.Data.Cycle + ULINT#2;
                MC_WriteParameterCycle := _AxisReference^.Data.Cycle ;
            END_IF;

            IF Execute THEN
                IF State = UINT#0 THEN
                    Busy := TRUE;
                    Parametrization.Inputs.Enable := FALSE;
                    State := UINT#190;
                END_IF;
                IF State = UINT#190 THEN
                    Busy := TRUE;
                    Parametrization.Inputs.Enable := TRUE;
                    Parametrization.Inputs.ReadWrite   := TRUE;
                    Parametrization.Inputs.ParameterNo := TO_INT(ParameterNumber);
                    Parametrization.Inputs.Subindex    := 0;
                    Parametrization.Inputs.AxisNo  := BYTE#1;
                    Parametrization.Inputs.HardwareId  := _AxisReference^.HWIDs.HW_ModuleAccessPoint;
                    Parametrization.Inputs.ValueWriteLINT := Value;
                    IF Parametrization.Outputs.Done AND NOT Parametrization.Outputs.Error THEN
                        State := UINT#191;
                    END_IF;
                    IF Parametrization.Outputs.Error THEN
                        Messenger.Activate(         UINT#1611, eAxoMessageCategory#Error);
                        MC_WriteParameterErrorID := DINT#1611;
                        State := UINT#199;
                    END_IF;
                END_IF;
                IF State = UINT#191 THEN
                    Busy := TRUE;
                    Parametrization.Inputs.Enable := FALSE;
                    Parametrization.Inputs.ReadWrite   := FALSE;
                    IF  NOT Parametrization.Outputs.Done THEN
                        State := UINT#197;
                    END_IF;
                END_IF;
                IF State = UINT#197 THEN
                    Done := TRUE;
                    MC_WriteParameterCycle := ULINT#0;
                END_IF;
                IF State = UINT#199 THEN
                    MC_WriteParameterCycle := ULINT#0;
                    Error := TRUE;
                END_IF;

                IF State>=UINT#190 AND State<UINT#197 THEN
                    IF _AxisReference^.Data.Cycle <> MC_WriteParameterCycle THEN
                        _AxisReference^.Data.Cycle := _AxisReference^.Data.Cycle - ULINT#1;
                        State := UINT#199;
                    END_IF;
                END_IF;
            END_IF;

            IF THIS.AxoWriteParameter_Task.DoneReached() THEN
                _AxisReference^.Status.CurrentMotionTaskId := AXOpen.Components.Drives.eAxoMotionTaskId#Axo_Done;
                MC_WriteParameterErrorID := DINT#0;
                // MC_WriteParameterCycle := ULINT#0;
                State := UINT#0;
            END_IF;

            IF THIS.AxoWriteParameter_Task.RestoreTriggered() AND State>=UINT#190 AND State<=UINT#199 THEN
                _AxisReference^.Status.CurrentMotionTaskId := AXOpen.Components.Drives.eAxoMotionTaskId#Axo_None;
                MC_WriteParameterErrorID := DINT#0;
                MC_WriteParameterCycle := ULINT#0;
                State := UINT#0;
            END_IF;

            ErrorID := MC_WriteParameterErrorID;
            MC_WriteParameterExecute_PV := Execute;
        END_METHOD

        ///<summary>
        /// This method modifies the value of a vendor specific parameter of type Real.
        ///</summary>
        VAR INTERNAL
            MC_WriteRealParameterExecute_PV     : 	BOOL := FALSE;		//Enable - previous value
            MC_WriteRealParameterErrorID        : 	DINT;
            MC_WriteRealParameterCycle			: 	ULINT;
        END_VAR
        METHOD PUBLIC OVERRIDE MC_WriteRealParameter
            VAR_INPUT
                AxisRef         :   AXOpen.Components.Abstractions.Drives.IAxoAxisReference;
                Execute         :   BOOL;                       //  Write the value of the parameter at rising edge
                ParameterNumber :   DINT;                       //  Number of the parameter (correspondence between number andparameter is specified in the table above)
                Value           :   REAL;                       //  New value of the specified parameter
                ExecutionMode   :   AXOpen.Components.Abstractions.Drives.eAxoExecutionMode;          //  Defines the chronological sequence of the method.
            END_VAR
            VAR_OUTPUT
                Done            :   BOOL;                       //  Parameter successfully written
                Busy            :   BOOL;                       //  The method is not finished and new output values are to be expected.
                Error           :   BOOL;                       //  Signals that an error has occurred within the method
                ErrorID         :   DINT;                       //  Error identification
            END_VAR
            VAR
                _AxisReference :  REF_TO AXOpen.Components.Festo.Drives.AxoCmmtAsAxisReference;
                Dummy : BOOL;
            END_VAR

            _AxisReference ?= AxisRef;

            IF(_AxisReference = NULL) THEN
                Messenger.Activate(     UINT#1620, eAxoMessageCategory#ProgrammingError);
                DriveStatus.Error.Id := UINT#1620;
                RETURN;
            END_IF;

            IF THIS.AxoWriteRealParameter_Task.StartTriggered()  THEN
                _AxisReference^.Status.CurrentMotionTaskId := AXOpen.Components.Drives.eAxoMotionTaskId#Axo_WriteRealParameter;
            END_IF;

            IF Execute AND NOT MC_WriteRealParameterExecute_PV AND State = UINT#0 THEN
                _AxisReference^.Data.Cycle := _AxisReference^.Data.Cycle + ULINT#2;
                MC_WriteRealParameterCycle := _AxisReference^.Data.Cycle ;
            END_IF;

            IF Execute THEN
                IF State = UINT#0 THEN
                    Busy := TRUE;
                    Parametrization.Inputs.Enable := FALSE;
                    State := UINT#200;
                END_IF;
                IF State = UINT#200 THEN
                    Busy := TRUE;
                    Parametrization.Inputs.Enable := TRUE;
                    Parametrization.Inputs.ReadWrite   := TRUE;
                    Parametrization.Inputs.ParameterNo := TO_INT(ParameterNumber);
                    Parametrization.Inputs.Subindex    := 0;
                    Parametrization.Inputs.AxisNo  := BYTE#1;
                    Parametrization.Inputs.HardwareId  := _AxisReference^.HWIDs.HW_ModuleAccessPoint;
                    Parametrization.Inputs.ValueWriteREAL := Value;
                    IF Parametrization.Outputs.Done AND NOT Parametrization.Outputs.Error THEN
                        State := UINT#201;
                    END_IF;
                    IF Parametrization.Outputs.Error THEN
                        Messenger.Activate(             UINT#1621, eAxoMessageCategory#Error);
                        MC_WriteRealParameterErrorID := DINT#1621;
                        State := UINT#209;
                    END_IF;
                END_IF;
                IF State = UINT#201 THEN
                    Busy := TRUE;
                    Parametrization.Inputs.Enable := FALSE;
                    Parametrization.Inputs.ReadWrite   := FALSE;
                    IF  NOT Parametrization.Outputs.Done THEN
                        State := UINT#207;
                    END_IF;
                END_IF;
                IF State = UINT#207 THEN
                    Done := TRUE;
                    MC_WriteRealParameterCycle := ULINT#0;
                END_IF;
                IF State = UINT#209 THEN
                    MC_WriteRealParameterCycle := ULINT#0;
                    Error := TRUE;
                END_IF;

                IF State>=UINT#200 AND State<UINT#207 THEN
                    IF _AxisReference^.Data.Cycle <> MC_WriteRealParameterCycle THEN
                        _AxisReference^.Data.Cycle := _AxisReference^.Data.Cycle - ULINT#1;
                        State := UINT#209;
                    END_IF;
                END_IF;
            END_IF;

            IF THIS.AxoWriteRealParameter_Task.DoneReached() THEN
                _AxisReference^.Status.CurrentMotionTaskId := AXOpen.Components.Drives.eAxoMotionTaskId#Axo_Done;
                MC_WriteRealParameterErrorID := DINT#0;
                // MC_WriteRealParameterCycle := ULINT#0;
                State := UINT#0;
            END_IF;

            IF THIS.AxoWriteRealParameter_Task.RestoreTriggered() AND State>=UINT#200 AND State<=UINT#209 THEN
                _AxisReference^.Status.CurrentMotionTaskId := AXOpen.Components.Drives.eAxoMotionTaskId#Axo_None;
                MC_WriteRealParameterErrorID := DINT#0;
                MC_WriteRealParameterCycle := ULINT#0;
                State := UINT#0;
            END_IF;

            ErrorID := MC_WriteRealParameterErrorID;
            MC_WriteRealParameterExecute_PV := Execute;
        END_METHOD

        ///<summary>
        /// This method modifies the value of a vendor specific parameter of type BOOL.
        ///</summary>
        VAR INTERNAL
            MC_WriteBoolParameterExecute_PV     : 	BOOL := FALSE;		//Enable - previous value
            MC_WriteBoolParameterErrorID        : 	DINT;
            MC_WriteBoolParameterCycle			: 	ULINT;
        END_VAR
        METHOD PUBLIC OVERRIDE MC_WriteBoolParameter
            VAR_INPUT
                AxisRef         :   AXOpen.Components.Abstractions.Drives.IAxoAxisReference;
                Execute         :   BOOL;                       //  Write the value of the parameter at rising edge
                ParameterNumber :   DINT;                       //  Number of the parameter (correspondence between number andparameter is specified in the table above)
                Value           :   BOOL;                       //  New value of the specified parameter
                ExecutionMode   :   AXOpen.Components.Abstractions.Drives.eAxoExecutionMode;          //  Defines the chronological sequence of the method.
            END_VAR
            VAR_OUTPUT
                Done            :   BOOL;                       //  Parameter successfully written
                Busy            :   BOOL;                       //  The method is not finished and new output values are to be expected.
                Error           :   BOOL;                       //  Signals that an error has occurred within the method
                ErrorID         :   DINT;                       //  Error identification
            END_VAR
            VAR
                _AxisReference :  REF_TO AXOpen.Components.Festo.Drives.AxoCmmtAsAxisReference;
                Dummy : BOOL;
            END_VAR

            _AxisReference ?= AxisRef;

            IF(_AxisReference = NULL) THEN
                Messenger.Activate(     UINT#1630, eAxoMessageCategory#ProgrammingError);
                DriveStatus.Error.Id := UINT#1630;
                RETURN;
            END_IF;

            IF THIS.AxoWriteBoolParameter_Task.StartTriggered()  THEN
                _AxisReference^.Status.CurrentMotionTaskId := AXOpen.Components.Drives.eAxoMotionTaskId#Axo_WriteBoolParameter;
            END_IF;

            IF Execute AND NOT MC_WriteBoolParameterExecute_PV AND State = UINT#0 THEN
                _AxisReference^.Data.Cycle := _AxisReference^.Data.Cycle + ULINT#2;
                MC_WriteBoolParameterCycle := _AxisReference^.Data.Cycle ;
            END_IF;

            IF Execute THEN
                IF State = UINT#0 THEN
                    Busy := TRUE;
                    Parametrization.Inputs.Enable := FALSE;
                    State := UINT#210;
                END_IF;
                IF State = UINT#210 THEN
                    Busy := TRUE;
                    Parametrization.Inputs.Enable := TRUE;
                    Parametrization.Inputs.ReadWrite   := TRUE;
                    Parametrization.Inputs.ParameterNo := TO_INT(ParameterNumber);
                    Parametrization.Inputs.Subindex    := 0;
                    Parametrization.Inputs.AxisNo  := BYTE#1;
                    Parametrization.Inputs.HardwareId  := _AxisReference^.HWIDs.HW_ModuleAccessPoint;
                    Parametrization.Inputs.ValueWriteBOOL := Value;
                    IF Parametrization.Outputs.Done AND NOT Parametrization.Outputs.Error THEN
                        State := UINT#211;
                    END_IF;
                    IF Parametrization.Outputs.Error THEN
                        Messenger.Activate(             UINT#1631, eAxoMessageCategory#Error);
                        MC_WriteBoolParameterErrorID := DINT#1631;
                        State := UINT#219;
                    END_IF;
                END_IF;
                IF State = UINT#211 THEN
                    Busy := TRUE;
                    Parametrization.Inputs.Enable := FALSE;
                    Parametrization.Inputs.ReadWrite   := FALSE;
                    IF  NOT Parametrization.Outputs.Done THEN
                        State := UINT#217;
                    END_IF;
                END_IF;
                IF State = UINT#217 THEN
                    Done := TRUE;
                    MC_WriteBoolParameterCycle := ULINT#0;
                END_IF;
                IF State = UINT#219 THEN
                    MC_WriteBoolParameterCycle := ULINT#0;
                    Error := TRUE;
                END_IF;

                IF State>=UINT#210 AND State<UINT#217 THEN
                    IF _AxisReference^.Data.Cycle <> MC_WriteBoolParameterCycle THEN
                        _AxisReference^.Data.Cycle := _AxisReference^.Data.Cycle - ULINT#1;
                        State := UINT#219;
                    END_IF;
                END_IF;
            END_IF;

            IF THIS.AxoWriteBoolParameter_Task.DoneReached() THEN
                _AxisReference^.Status.CurrentMotionTaskId := AXOpen.Components.Drives.eAxoMotionTaskId#Axo_Done;
                MC_WriteBoolParameterErrorID := DINT#0;
                // MC_WriteBoolParameterCycle := ULINT#0;
                State := UINT#0;
            END_IF;

            IF THIS.AxoWriteBoolParameter_Task.RestoreTriggered() AND State>=UINT#210 AND State<=UINT#219 THEN
                _AxisReference^.Status.CurrentMotionTaskId := AXOpen.Components.Drives.eAxoMotionTaskId#Axo_None;
                MC_WriteBoolParameterErrorID := DINT#0;
                MC_WriteBoolParameterCycle := ULINT#0;
                State := UINT#0;
            END_IF;

            ErrorID := MC_WriteBoolParameterErrorID;
            MC_WriteBoolParameterExecute_PV := Execute;
        END_METHOD

        ///<summary>
        /// This method gives access to the value of the input, referenced by the datatype MC_INPUT_REF.
        /// It provides the value of the referenced input (BOOL).
        ///</summary>
        VAR INTERNAL
            MC_ReadDigitalInputEnable_PV        : 	BOOL := FALSE;		//Enable - previous value
            MC_ReadDigitalInputErrorID          : 	DINT;
            MC_ReadDigitalInputCycle			: 	ULINT;
            MC_ReadDigitalInputValue			: 	BOOL;
            MC_ReadDigitalInputValid			: 	BOOL;
        END_VAR
        METHOD PUBLIC OVERRIDE MC_ReadDigitalInput
            VAR_INPUT
                AxisRef         :   AXOpen.Components.Abstractions.Drives.IAxoAxisReference;
                Enable          :   BOOL;                       //  Get the value of the selected input signal continuously while enabled
                InputNumber     :   INT;                        //  Selects the input. Can be part of MC_INPUT_REF, if only one single input is referenced.
            END_VAR
            VAR_OUTPUT
                Valid           :   BOOL;                       //  A valid output is available at the method
                Busy            :   BOOL;                       //  The method is not finished and new output values are to be expected
                Error           :   BOOL;                       //  Signals that an error has occurred within the method
                ErrorID         :   DINT;                       //  Error identification
                Value           :   BOOL;                       //  The value of the selected input signal
            END_VAR
            VAR
                _AxisReference :  REF_TO AXOpen.Components.Festo.Drives.AxoCmmtAsAxisReference;
                Dummy : BOOL;
            END_VAR

            _AxisReference ?= AxisRef;

            IF(_AxisReference = NULL) THEN
                Messenger.Activate(     UINT#1640, eAxoMessageCategory#ProgrammingError);
                DriveStatus.Error.Id := UINT#1640;
                RETURN;
            END_IF;

            IF(InputNumber < 0 OR InputNumber > 64) THEN   //  TODO check the min max input number
                Messenger.Activate(     UINT#1641, eAxoMessageCategory#ProgrammingError);
                DriveStatus.Error.Id := UINT#1641;
                RETURN;
            END_IF;

            IF Enable AND NOT MC_ReadDigitalInputEnable_PV AND State = UINT#0 THEN
                _AxisReference^.Status.CurrentMotionTaskId := AXOpen.Components.Drives.eAxoMotionTaskId#Axo_ReadDigitalInput;
                _AxisReference^.Data.Cycle := _AxisReference^.Data.Cycle + ULINT#2;
                MC_ReadDigitalInputCycle := _AxisReference^.Data.Cycle ;
            END_IF;

            IF Enable THEN
                IF State = UINT#0 THEN
                    Busy := TRUE;
                    MC_ReadDigitalInputErrorID := DINT#0;
                    Parametrization.Inputs.Enable := FALSE;
                    State := UINT#220;
                END_IF;
                IF State = UINT#220 THEN
                    Busy := TRUE;
                    Parametrization.Inputs.Enable := TRUE;
                    Parametrization.Inputs.ReadWrite   := FALSE;
                    IF InputNumber>= 0 AND InputNumber < 32 THEN
                        Parametrization.Inputs.ParameterNo := 2888;  //X1A
                    ELSIF InputNumber>= 32 AND InputNumber < 64 THEN
                        Parametrization.Inputs.ParameterNo := 2889;  //X1C
                    END_IF;
                    Parametrization.Inputs.Subindex    := 0;
                    Parametrization.Inputs.AxisNo  := BYTE#1;
                    Parametrization.Inputs.HardwareId  := _AxisReference^.HWIDs.HW_ModuleAccessPoint;
                    IF Parametrization.Outputs.Done AND NOT Parametrization.Outputs.Error THEN
                        MC_ReadDigitalInputValid := TRUE;
                        IF InputNumber>= 0 AND InputNumber < 32 THEN
                            MC_ReadDigitalInputValue := GetBit(TO_LWORD(Parametrization.Outputs.ValueReadLINT), TO_USINT(InputNumber)); //X1A
                        ELSIF InputNumber>= 32 AND InputNumber < 64 THEN
                            MC_ReadDigitalInputValue := GetBit(TO_LWORD(Parametrization.Outputs.ValueReadLINT), TO_USINT(InputNumber-INT#32)); //X1C
                        END_IF;
                        State := UINT#221;
                    END_IF;
                    IF Parametrization.Outputs.Error THEN
                        Messenger.Activate(             UINT#1642, eAxoMessageCategory#Error);
                        MC_ReadDigitalInputErrorID :=   DINT#1642;
                        State := UINT#229;
                    END_IF;
                END_IF;
                IF State = UINT#221 THEN
                    Busy := TRUE;
                    Parametrization.Inputs.Enable := FALSE;
                    Parametrization.Inputs.ReadWrite   := FALSE;
                    IF  NOT Parametrization.Outputs.Done THEN
                        State := UINT#220;
                    END_IF;
                END_IF;
                IF State = UINT#229 THEN
                    Error := TRUE;
                END_IF;

                IF State>=UINT#220 AND State<UINT#227 THEN
                    IF _AxisReference^.Data.Cycle <> MC_ReadDigitalInputCycle THEN
                        _AxisReference^.Data.Cycle := _AxisReference^.Data.Cycle - ULINT#1;
                        State := UINT#229;
                    END_IF;
                END_IF;
            END_IF;

            IF NOT Enable AND MC_ReadDigitalInputEnable_PV  THEN
                _AxisReference^.Status.CurrentMotionTaskId := AXOpen.Components.Drives.eAxoMotionTaskId#Axo_None;
                MC_ReadDigitalInputErrorID := DINT#0;
                MC_ReadDigitalInputCycle := ULINT#0;
                MC_ReadDigitalInputValid := FALSE;
                MC_ReadDigitalInputValue := FALSE;
                State := UINT#0;
            END_IF;

            ErrorID := MC_ReadDigitalInputErrorID;
            Valid := MC_ReadDigitalInputValid;
            Value := MC_ReadDigitalInputValue;
            MC_ReadDigitalInputEnable_PV := Enable;
        END_METHOD

        ///<summary>
        /// This method provides access to the value of a digital output, referenced by the datatype MC_OUTPUT_REF.
        /// It provides the value of the referenced output (BOOL).
        ///</summary>
        VAR INTERNAL
            MC_ReadDigitalOutputEnable_PV        : 	BOOL := FALSE;		//Enable - previous value
            MC_ReadDigitalOutputErrorID          : 	DINT;
            MC_ReadDigitalOutputCycle			: 	ULINT;
            MC_ReadDigitalOutputValue			: 	BOOL;
            MC_ReadDigitalOutputValid			: 	BOOL;
        END_VAR
        METHOD PUBLIC OVERRIDE MC_ReadDigitalOutput
            VAR_INPUT
                AxisRef         :   AXOpen.Components.Abstractions.Drives.IAxoAxisReference;
                Enable          :   BOOL;                       //  Get the value of the selected output signal continuously while enabled
                OutputNumber    :   INT;                        //  Selects the output. Can be part of MC_OUTPUT_REF, if only one single output is referenced.
            END_VAR
            VAR_OUTPUT
                Valid           :   BOOL;                       //  A valid output is available at the method
                Busy            :   BOOL;                       //  The method is not finished and new output values are to be expected
                Error           :   BOOL;                       //  Signals that an error has occurred within the method
                ErrorID         :   DINT;                       //  Error identification
                Value           :   BOOL;                       //  The value of the selected output signal
            END_VAR
            VAR
                _AxisReference :  REF_TO AXOpen.Components.Festo.Drives.AxoCmmtAsAxisReference;
                Dummy : BOOL;
            END_VAR

            _AxisReference ?= AxisRef;

            IF(_AxisReference = NULL) THEN
                Messenger.Activate(     UINT#1650, eAxoMessageCategory#ProgrammingError);
                DriveStatus.Error.Id := UINT#1650;
                RETURN;
            END_IF;

            IF(OutputNumber < 0 OR OutputNumber >256) THEN   //  TODO check the min max input number
                Messenger.Activate(     UINT#1651, eAxoMessageCategory#ProgrammingError);
                DriveStatus.Error.Id := UINT#1651;
                RETURN;
            END_IF;

            IF Enable AND NOT MC_ReadDigitalOutputEnable_PV AND State = UINT#0 THEN
                _AxisReference^.Status.CurrentMotionTaskId := AXOpen.Components.Drives.eAxoMotionTaskId#Axo_ReadDigitalOutput;
                _AxisReference^.Data.Cycle := _AxisReference^.Data.Cycle + ULINT#2;
                MC_ReadDigitalOutputCycle := _AxisReference^.Data.Cycle ;
            END_IF;

            IF Enable THEN
                IF State = UINT#0 THEN
                    Busy := TRUE;
                    MC_ReadDigitalOutputErrorID := DINT#0;
                    Parametrization.Inputs.Enable := FALSE;
                    State := UINT#230;
                END_IF;
                IF State = UINT#230 THEN
                    Busy := TRUE;
                    Parametrization.Inputs.Enable := TRUE;
                    Parametrization.Inputs.ReadWrite   := FALSE;
                    Parametrization.Inputs.ParameterNo := 2888;
                    Parametrization.Inputs.Subindex    := 0;
                    Parametrization.Inputs.AxisNo  := BYTE#1;
                    Parametrization.Inputs.HardwareId  := _AxisReference^.HWIDs.HW_ModuleAccessPoint;
                    IF Parametrization.Outputs.Done AND NOT Parametrization.Outputs.Error THEN
                        MC_ReadDigitalOutputValid := TRUE;
                        MC_ReadDigitalOutputValue := GetBit(TO_LWORD(Parametrization.Outputs.ValueReadLINT), TO_USINT(OutputNumber));
                        State := UINT#231;
                    END_IF;
                    IF Parametrization.Outputs.Error THEN
                        Messenger.Activate(             UINT#1652, eAxoMessageCategory#Error);
                        MC_ReadDigitalOutputErrorID :=  DINT#1652;
                        State := UINT#239;
                    END_IF;
                END_IF;
                IF State = UINT#231 THEN
                    Busy := TRUE;
                    Parametrization.Inputs.Enable := FALSE;
                    Parametrization.Inputs.ReadWrite   := FALSE;
                    IF  NOT Parametrization.Outputs.Done THEN
                        State := UINT#230;
                    END_IF;
                END_IF;
                IF State = UINT#239 THEN
                    Error := TRUE;
                END_IF;

                IF State>=UINT#230 AND State<UINT#237 THEN
                    IF _AxisReference^.Data.Cycle <> MC_ReadDigitalOutputCycle THEN
                        _AxisReference^.Data.Cycle := _AxisReference^.Data.Cycle - ULINT#1;
                        State := UINT#239;
                    END_IF;
                END_IF;
            END_IF;

            IF NOT Enable AND MC_ReadDigitalOutputEnable_PV  THEN
                _AxisReference^.Status.CurrentMotionTaskId := AXOpen.Components.Drives.eAxoMotionTaskId#Axo_None;
                MC_ReadDigitalOutputErrorID := DINT#0;
                MC_ReadDigitalOutputCycle := ULINT#0;
                MC_ReadDigitalOutputValid := FALSE;
                MC_ReadDigitalOutputValue := FALSE;
                State := UINT#0;
            END_IF;

            ErrorID := MC_ReadDigitalOutputErrorID;
            Valid := MC_ReadDigitalOutputValid;
            Value := MC_ReadDigitalOutputValue;
            MC_ReadDigitalOutputEnable_PV := Enable;
        END_METHOD

        ///<summary>
        /// This method writes a value to the output referenced by the argument ‘Output’ once (with rising edge of Execute)
        ///</summary>
        VAR INTERNAL
            MC_WriteDigitalOutputExecute_PV     : 	BOOL := FALSE;		//Enable - previous value
            MC_WriteDigitalOutputErrorID        : 	DINT;
            MC_WriteDigitalOutputCycle			: 	ULINT;
        END_VAR
        METHOD PUBLIC OVERRIDE MC_WriteDigitalOutput
            VAR_INPUT
                AxisRef         :   AXOpen.Components.Abstractions.Drives.IAxoAxisReference;
                Execute         :   BOOL;                       //  Write the value of the selected output
                OutputNumber    :   INT;                        //  Selects the output. Can be part of MC_OUTPUT_REF, if only one single output is referenced.
                Value           :   BOOL;                       //  The value of the selected output signal
                ExecutionMode   :   AXOpen.Components.Abstractions.Drives.eAxoExecutionMode;          //  Defines the chronological sequence of the method.
            END_VAR
            VAR_OUTPUT
                Done            :   BOOL;                       //  Writing of the output signal value is done
                Busy            :   BOOL;                       //  The method is not finished and new output values are to be expected.
                Error           :   BOOL;                       //  Signals that an error has occurred within the method
                ErrorID         :   DINT;                       //  Error identification
            END_VAR
            VAR
                _AxisReference :  REF_TO AXOpen.Components.Festo.Drives.AxoCmmtAsAxisReference;
                Dummy : BOOL;
                Valid_          :   BOOL;
                Error_          :   BOOL;
                ErrorID_        :   WORD;
            END_VAR

            _AxisReference ?= AxisRef;

            IF(_AxisReference = NULL) THEN
                Messenger.Activate(     UINT#1660, eAxoMessageCategory#ProgrammingError);
                DriveStatus.Error.Id := UINT#1660;
                RETURN;
            END_IF;

            IF(OutputNumber < 0 OR OutputNumber >256) THEN   //  TODO check the min max input number
                Messenger.Activate(     UINT#1661, eAxoMessageCategory#ProgrammingError);
                DriveStatus.Error.Id := UINT#1661;
                RETURN;
            END_IF;

            IF THIS.AxoWriteDigitalOutput_Task.StartTriggered()  THEN
                _AxisReference^.Status.CurrentMotionTaskId := AXOpen.Components.Drives.eAxoMotionTaskId#Axo_WriteDigitalOutput;
            END_IF;

            IF Execute AND NOT MC_WriteDigitalOutputExecute_PV AND State = UINT#0 THEN
                _AxisReference^.Data.Cycle := _AxisReference^.Data.Cycle + ULINT#2;
                MC_WriteDigitalOutputCycle := _AxisReference^.Data.Cycle ;
            END_IF;

            IF Execute THEN
                IF State = UINT#0 THEN
                    Busy := TRUE;
                    Parametrization.Inputs.Enable := FALSE;
                    State := UINT#240;
                    //Remove after implementation on the drive side
                    State := UINT#249;
                    Messenger.Activate(             UINT#1662, eAxoMessageCategory#ProgrammingError);
                    MC_WriteDigitalOutputErrorID := DINT#1662;
                END_IF;
                IF State = UINT#240 THEN
                    Busy := TRUE;
                    Parametrization.Inputs.Enable := TRUE;
                    Parametrization.Inputs.ReadWrite   := TRUE;
                    Parametrization.Inputs.ParameterNo := 0;
                    Parametrization.Inputs.Subindex    := 0;
                    Parametrization.Inputs.AxisNo  := BYTE#1;
                    Parametrization.Inputs.HardwareId  := _AxisReference^.HWIDs.HW_ModuleAccessPoint;
                    Parametrization.Inputs.ValueWriteBOOL := Value;
                    IF Parametrization.Outputs.Done AND NOT Parametrization.Outputs.Error THEN
                        State := UINT#241;
                    END_IF;
                    IF Parametrization.Outputs.Error THEN
                        Messenger.Activate(             UINT#1663, eAxoMessageCategory#Error);
                        MC_WriteDigitalOutputErrorID := DINT#1663;
                        State := UINT#249;
                    END_IF;
                END_IF;
                IF State = UINT#241 THEN
                    Busy := TRUE;
                    Parametrization.Inputs.Enable := FALSE;
                    Parametrization.Inputs.ReadWrite   := FALSE;
                    IF  NOT Parametrization.Outputs.Done THEN
                        State := UINT#247;
                    END_IF;
                END_IF;
                IF State = UINT#247 THEN
                    Done := TRUE;
                    MC_WriteDigitalOutputCycle := ULINT#0;
                END_IF;
                IF State = UINT#249 THEN
                    MC_WriteDigitalOutputCycle := ULINT#0;
                    Error := TRUE;
                END_IF;

                IF State>=UINT#240 AND State<UINT#247 THEN
                    IF _AxisReference^.Data.Cycle <> MC_WriteDigitalOutputCycle THEN
                        _AxisReference^.Data.Cycle := _AxisReference^.Data.Cycle - ULINT#1;
                        State := UINT#249;
                    END_IF;
                END_IF;
            END_IF;

            IF THIS.AxoWriteDigitalOutput_Task.DoneReached() THEN
                _AxisReference^.Status.CurrentMotionTaskId := AXOpen.Components.Drives.eAxoMotionTaskId#Axo_Done;
                MC_WriteDigitalOutputErrorID := DINT#0;
                // MC_WriteDigitalOutputCycle := ULINT#0;
                State := UINT#0;
            END_IF;

            IF THIS.AxoWriteDigitalOutput_Task.RestoreTriggered() AND State>=UINT#240 AND State<=UINT#249 THEN
                _AxisReference^.Status.CurrentMotionTaskId := AXOpen.Components.Drives.eAxoMotionTaskId#Axo_None;
                MC_WriteDigitalOutputErrorID := DINT#0;
                MC_WriteDigitalOutputCycle := ULINT#0;
                State := UINT#0;
            END_IF;

            ErrorID := MC_WriteDigitalOutputErrorID;
            MC_WriteDigitalOutputExecute_PV := Execute;

        END_METHOD

        ///<summary>
        /// This method returns the actual position.
        ///<summary>
        METHOD PUBLIC OVERRIDE MC_ReadActualPosition
             VAR_INPUT
                AxisRef         :   AXOpen.Components.Abstractions.Drives.IAxoAxisReference;
                Enable          :   BOOL;                       //  Get the value of the parameter continuously while enabled
            END_VAR
            VAR_OUTPUT
                Valid           :   BOOL;                       //  A valid output is available at the method
                Busy            :   BOOL;                       //  The method is not finished and new output values are to be expected
                Error           :   BOOL;                       //  Signals that an error has occurred within the method
                ErrorID         :   DINT;                       //  Error identification
                Position        :   LREAL;                       //  New absolute position (in axis’ unit [u])
            END_VAR
            VAR
                _AxisReference :  REF_TO AXOpen.Components.Festo.Drives.AxoCmmtAsAxisReference;
                Dummy : BOOL;
            END_VAR

            _AxisReference ?= AxisRef;

            IF(_AxisReference = NULL) THEN
                Messenger.Activate(     UINT#1670, eAxoMessageCategory#ProgrammingError);
                DriveStatus.Error.Id := UINT#1670;
                RETURN;
            END_IF;

            IF Enable THEN
                THIS.UpdateInputs(AxisRef);
                Valid := TRUE;
                Position := THIS.ActualPosition;
            END_IF;
        END_METHOD

        ///<summary>
        /// This method returns the value of the actual velocity as long as ‘Enable’ is set. ‘Valid’ is true when the
        /// dataoutput ‘Velocity’ is valid. If ‘Enable’ is Reset, the data loses its validity, and all outputs are reset,
        /// no matter if new data is available.
        ///<summary>
        METHOD PUBLIC OVERRIDE MC_ReadActualVelocity
            VAR_INPUT
                AxisRef         :   AXOpen.Components.Abstractions.Drives.IAxoAxisReference;
                Enable          :   BOOL;                       //  Get the value of the parameter continuously while enabled
            END_VAR
            VAR_OUTPUT
                Valid           :   BOOL;                       //  A valid output is available at the method
                Busy            :   BOOL;                       //  The method is not finished and new output values are to be expected
                Error           :   BOOL;                       //  Signals that an error has occurred within the method
                ErrorID         :   DINT;                       //  Error identification
                Velocity        :   LREAL;                       //  The value of the actual velocity (in axis’ unit [u/s])
            END_VAR
            VAR
                _AxisReference :  REF_TO AXOpen.Components.Festo.Drives.AxoCmmtAsAxisReference;
                Dummy : BOOL;
            END_VAR

            _AxisReference ?= AxisRef;

            IF(_AxisReference = NULL) THEN
                Messenger.Activate(     UINT#1680, eAxoMessageCategory#ProgrammingError);
                DriveStatus.Error.Id := UINT#1680;
                RETURN;
            END_IF;

            IF Enable THEN
                THIS.UpdateInputs(AxisRef);
                Valid := TRUE;
                Velocity := THIS.ActualVelocity;
            END_IF;
        END_METHOD

        ///<summary>
        /// This method returns the value of the actual torque or force as long as ‘Enable’ is set. ‘Valid’ is true when the
        /// data-output ‘Torque’ is valid. If ‘Enable’ is Reset, the data loses its validity, and ‘Valid’ is also reset,
        /// no matter if new data is available.
        ///<summary>
        METHOD PUBLIC OVERRIDE MC_ReadActualTorque
            VAR_INPUT
                AxisRef         :   AXOpen.Components.Abstractions.Drives.IAxoAxisReference;
                Enable          :   BOOL;                       //  Get the value of the parameter continuously while enabled
            END_VAR
            VAR_OUTPUT
                Valid           :   BOOL;                       //  A valid output is available at the method
                Busy            :   BOOL;                       //  The method is not finished and new output values are to be expected
                Error           :   BOOL;                       //  Signals that an error has occurred within the method
                ErrorID         :   DINT;                       //  Error identification
                Torque          :   LREAL;                       //  The value of the actual torque or force (in technical units)
            END_VAR
            VAR
                _AxisReference :  REF_TO AXOpen.Components.Festo.Drives.AxoCmmtAsAxisReference;
                Dummy : BOOL;
            END_VAR
